(* CODESYS project Traffic_lights.project
   Title: Traffic_lights_ordinary
   Version: 0.0.0.0
   Author: Armin

Project tree, tasks and I/O mapping:
  MyController : TM241CE24T/U, Schneider Electric, order no. TM241CE24T/U, version 4.0.6.18
    application Application
      task MAST (cyclic, interval 20 ms, priority 15, watchdog 100 ms x 1) calls POU, POU_1
      global variables GVL
      Symbols
      program POU [SFC]: Sporedna_active, Sporedna_entry, Glavna_active, Glavna_entry, SveZuto_active, SveZuto_entry, SveZuto_exit, SamoGlavna_entry, SamoGlavna_active, SamoGlavna_exit, SamoSporedna_active, SamoSporedna_entry, SamoSporedna_exit
      program POU_1 [ST]
    DI : Digital Inputs, Schneider Electric, version 4.0.6.18
        input  iwDI_IW0 : WORD  // IW0
        input  ibDI_IB1 : BYTE  // IB1
    DQ : Digital Outputs, Schneider Electric, version 4.0.6.18
        output qwDQ_QW0 : WORD  // QW0
        output qbDQ_QB1 : BYTE  // QB1
    Counters : Counters, Schneider Electric, version 4.0.6.18
    Pulse_Generators : Pulse Generators, Schneider Electric, version 4.0.6.18
    Cartridge_1 : Cartridge, Schneider Electric, version 4.0.6.18
    IO_Bus : IO bus - TM3, Schneider Electric, version 4.0.6.18
    COM_Bus : COM bus, Schneider Electric, version 4.0.6.18
    Ethernet_1 : Ethernet Network, Schneider Electric, version 4.0.6.18
    Serial_Line_1 : Serial line, Schneider Electric, version 4.0.6.18
      SoMachine_Network_Manager : SoMachine-Network Manager, Schneider Electric, version 4.0.0.2
    Serial_Line_2 : Serial line, Schneider Electric, version 4.0.6.18
      Modbus_Manager : Modbus Manager, Schneider Electric, version 4.0.0.2
  XBTGT7340 : XBTGT7340, Schneider Electric, order no. XBTGT7340, version 3.5.3.54
    HMI Application
    COM1
      SoMachine_Network_Manager1 : SoMachine-Network Manager, Schneider Electric, version 4.0.0.2
    COM2
      SoMachine_Network_Manager2 : SoMachine-Network Manager, Schneider Electric, version 4.0.0.2
    Ethernet
      SoMachine_Network_Manager3 : SoMachine-Network Manager, Schneider Electric, version 4.0.0.2
    USB
      SoMachine_Network_Manager4 : SoMachine-Network Manager, Schneider Electric, version 4.0.0.2
  Vijeo Designer Project Container Data
  Vijeo Designer Project Container
*)

// MyController/Application/GVL
VAR_GLOBAL
	sifra: INT;
	stanje: BOOL;
	T1: TP;
	potvrdi: BOOL;
	vratiNaNulu: BOOL;
	
	proba: BOOL;
	noviStart: BOOL;
	noviStop: BOOL;
	
	ispis: INT;
	Glavna_dodatno_vrijeme: INT := 0;
	Sporedna_dodatno_vrijeme: INT := 0;
	
	Vrijeme_glavne_trake: INT := 65;
	Vrijeme_sporedne_trake: INT := 15;
	
	Inicijalno_vrijeme_glavne_trake: INT := 65;
	Inicijalno_vrijeme_sporedne_trake: INT := 15;
	
	Glavna_gornja_granica: INT := 120;
	Glavna_donja_granica: INT := 60;
	
	Sporedna_gornja_granica: INT := 120;
	Sporedna_donja_granica: INT := 12;
	
	Greska_unos_vremena1: BOOL;
	Greska_unos_vremena2: BOOL;
	
	Zuto_FF: RS;
	Zuto_FF_set: BOOL;
	Zuto_FF_reset: BOOL;
	
	save_glavna_vrijeme: INT;
	save_sporedna_vrijeme: INT;
	
	klik_na_glavna_save: BOOL;
	klik_na_sporedna_save: BOOL;
	uso1: BOOL;
	uso2: BOOL;
	proso1: BOOL := 1;
	
	Glavna_FF: RS;
	Glavna_FF_set: BOOL;
	Glavna_FF_reset: BOOL;
	
	Sporedna_FF: RS;
	Sporedna_FF_set: BOOL;
	Sporedna_FF_reset: BOOL;
	
	resetuj: BOOL;
END_VAR

// MyController/Application/POU
PROGRAM POU
VAR
	okidac: BOOL;
	timer: TOF;
	Glavna4_G: BOOL;
	Glavna4_Y: BOOL;
	Glavna4_R: BOOL;
	Glavna4_lijevo_G: BOOL;
	Glavna4_lijevo_Y: BOOL;
	Glavna4_lijevo_R: BOOL;
	Glavna5_G: BOOL;
	Glavna5_Y: BOOL;
	Glavna5_R: BOOL;
	Glavna5_lijevo_G: BOOL;
	Glavna5_lijevo_Y: BOOL;
	Glavna5_lijevo_R: BOOL;
	Sporedna_G: BOOL;
	Sporedna_Y: BOOL;
	Sporedna_R: BOOL;
	Sporedna_blinkanje: BOOL;
	Glavna5_lijevo_blinkanje: BOOL;
	Glavna5_blinkanje: BOOL;
	Glavna4_lijevo_blinkanje: BOOL;
	Glavna4_blinkanje: BOOL;
	Tramvaj: BOOL;
	Glavna5_pjesaci: BOOL;
	Glavna5_pjesaci_preko: BOOL;
	// Trebao bi se ukljuciti odmah po ukljucenju crvenog na tom dijelu, sto nije slucaj u stvarnosti
	Glavna4_pjesaci: BOOL;
	Glavna4_pjesaci_preko: BOOL;
	Sporedna_jug_pjesaci: BOOL;
	// Trebalo bi se odmah ukljuciti cim se ukljuci zeleno na Glavna5, ovako ni pjesaci ni vozaci nisu sigurni ko treba da ide, jer se za zeleno pjesake ceka 4 sekunde od zelenog za vozace
	Sporedna_sjever_pjesaci: BOOL;
	Sve_zuto_blinkanje: BOOL;
END_VAR

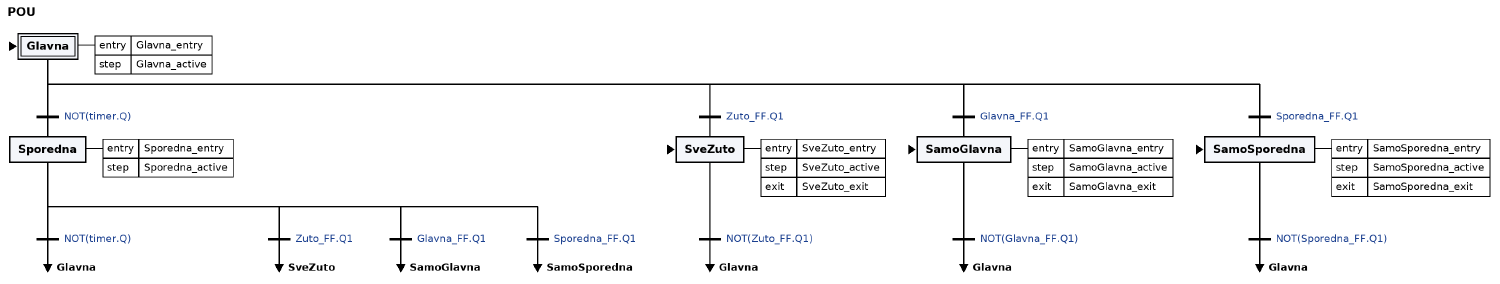
INITIAL_STEP Glavna:
    Glavna_entry(P1);  // entry action
    Glavna_active(N);  // step action
END_STEP
TRANSITION FROM Glavna TO Sporedna
    := NOT(timer.Q);
END_TRANSITION
STEP Sporedna:
    Sporedna_entry(P1);  // entry action
    Sporedna_active(N);  // step action
END_STEP
TRANSITION FROM Sporedna TO Glavna
    := NOT(timer.Q);
END_TRANSITION
TRANSITION FROM Sporedna TO SveZuto
    := Zuto_FF.Q1;
END_TRANSITION
TRANSITION FROM Sporedna TO SamoGlavna
    := Glavna_FF.Q1;
END_TRANSITION
TRANSITION FROM Sporedna TO SamoSporedna
    := Sporedna_FF.Q1;
END_TRANSITION
TRANSITION FROM Glavna TO SveZuto
    := Zuto_FF.Q1;
END_TRANSITION
STEP SveZuto:
    SveZuto_entry(P1);  // entry action
    SveZuto_active(N);  // step action
    SveZuto_exit(P0);  // exit action
END_STEP
TRANSITION FROM SveZuto TO Glavna
    := NOT(Zuto_FF.Q1);
END_TRANSITION
TRANSITION FROM Glavna TO SamoGlavna
    := Glavna_FF.Q1;
END_TRANSITION
STEP SamoGlavna:
    SamoGlavna_entry(P1);  // entry action
    SamoGlavna_active(N);  // step action
    SamoGlavna_exit(P0);  // exit action
END_STEP
TRANSITION FROM SamoGlavna TO Glavna
    := NOT(Glavna_FF.Q1);
END_TRANSITION
TRANSITION FROM Glavna TO SamoSporedna
    := Sporedna_FF.Q1;
END_TRANSITION
STEP SamoSporedna:
    SamoSporedna_entry(P1);  // entry action
    SamoSporedna_active(N);  // step action
    SamoSporedna_exit(P0);  // exit action
END_STEP
TRANSITION FROM SamoSporedna TO Glavna
    := NOT(Sporedna_FF.Q1);
END_TRANSITION

ACTION Sporedna_active:
timer(IN := okidac, PT := LINT_TO_TIME((Vrijeme_sporedne_trake - Inicijalno_vrijeme_sporedne_trake)*1000) + T#15S);
okidac := FALSE;

IF timer.ET > T#2S THEN
	Sporedna_R := 0;
	Sporedna_Y := 0;
	Sporedna_G := 1;
END_IF

IF timer.ET > T#3S THEN
	Glavna5_pjesaci_preko := 1;
	Glavna4_pjesaci_preko := 1;
END_IF

IF timer.ET > LINT_TO_TIME((Vrijeme_sporedne_trake - Inicijalno_vrijeme_sporedne_trake)*1000) + T#4S THEN
	Glavna4_pjesaci := 0;
END_IF

IF timer.ET > LINT_TO_TIME((Vrijeme_sporedne_trake - Inicijalno_vrijeme_sporedne_trake)*1000) + T#8S THEN
	Sporedna_blinkanje := 1;
END_IF

IF timer.ET > LINT_TO_TIME((Vrijeme_sporedne_trake - Inicijalno_vrijeme_sporedne_trake)*1000) + T#12S THEN
	Sporedna_blinkanje := 0;
	Sporedna_G := 0;
	Sporedna_Y := 1;
END_IF

IF timer.ET > LINT_TO_TIME((Vrijeme_sporedne_trake - Inicijalno_vrijeme_sporedne_trake)*1000) + T#13S THEN
	Glavna5_pjesaci_preko := 0;
	Glavna4_pjesaci_preko := 0;
END_IF

IF timer.ET > LINT_TO_TIME((Vrijeme_sporedne_trake - Inicijalno_vrijeme_sporedne_trake)*1000) + T#14S THEN
	Sporedna_Y := 0;
	Sporedna_R := 1;
END_IF
END_ACTION

ACTION Sporedna_entry:
okidac := TRUE;
Sporedna_R := 1;
Sporedna_Y := 1;
END_ACTION

ACTION Glavna_active:
timer(IN := okidac, PT := LINT_TO_TIME((Vrijeme_glavne_trake - Inicijalno_vrijeme_glavne_trake)*1000) + T#65S);
okidac := FALSE;

IF timer.ET > T#2S THEN
	Glavna4_Y := 1;
	Glavna4_lijevo_Y := 1;
END_IF

IF timer.ET > T#4S THEN
	Glavna4_R := 0;
	Glavna4_lijevo_R := 0;
	Glavna4_Y := 0;
	Glavna4_lijevo_Y := 0;
	Glavna4_G := 1;
	Glavna4_lijevo_G := 1;
END_IF

IF timer.ET > T#5S THEN
	Sporedna_jug_pjesaci := 1;
END_IF

IF timer.ET > T#10S THEN
	Glavna5_pjesaci := 0;
END_IF

IF timer.ET > T#13S THEN
	Glavna4_lijevo_blinkanje := 1;
END_IF

IF timer.ET > T#17S THEN
	Glavna4_lijevo_blinkanje := 0;
	Glavna4_lijevo_G := 0;
	Glavna4_lijevo_Y := 1;
END_IF

IF timer.ET > T#20S THEN
	Glavna4_lijevo_Y := 0;
	Glavna4_lijevo_R := 1;
END_IF

IF timer.ET > T#23S THEN
	Glavna5_Y := 1;
END_IF

IF timer.ET > T#25S THEN
	Glavna5_R := 0;
	Glavna5_Y := 0;
	Glavna5_G := 1;
	Tramvaj := 1;
END_IF

IF timer.ET > T#26S THEN
	Sporedna_sjever_pjesaci := 1;
END_IF

IF timer.ET > LINT_TO_TIME((Vrijeme_glavne_trake - Inicijalno_vrijeme_glavne_trake)*1000) + T#33S THEN
	Sporedna_jug_pjesaci := 0;
END_IF

IF timer.ET > LINT_TO_TIME((Vrijeme_glavne_trake - Inicijalno_vrijeme_glavne_trake)*1000) + T#40S THEN
	Glavna4_blinkanje := 1;
	Tramvaj := 0;
	Sporedna_sjever_pjesaci := 0;
END_IF

IF timer.ET > LINT_TO_TIME((Vrijeme_glavne_trake - Inicijalno_vrijeme_glavne_trake)*1000) + T#44S THEN
	Glavna4_blinkanje := 0;
	Glavna4_G := 0;
	Glavna4_Y := 1;
END_IF

IF timer.ET > LINT_TO_TIME((Vrijeme_glavne_trake - Inicijalno_vrijeme_glavne_trake)*1000) + T#47S THEN
	Glavna4_Y := 0;
	Glavna4_R := 1;
END_IF

IF timer.ET > LINT_TO_TIME((Vrijeme_glavne_trake - Inicijalno_vrijeme_glavne_trake)*1000) + T#48S THEN
	Glavna5_lijevo_Y := 1;
	Glavna4_pjesaci := 1;
END_IF

IF timer.ET > LINT_TO_TIME((Vrijeme_glavne_trake - Inicijalno_vrijeme_glavne_trake)*1000) + T#50S THEN
	Glavna5_lijevo_R := 0;
	Glavna5_lijevo_Y := 0;
	Glavna5_lijevo_G := 1;
END_IF

IF timer.ET > LINT_TO_TIME((Vrijeme_glavne_trake - Inicijalno_vrijeme_glavne_trake)*1000) + T#56S THEN
	Glavna5_lijevo_blinkanje := 1;
	Glavna5_blinkanje := 1;
END_IF

IF timer.ET > LINT_TO_TIME((Vrijeme_glavne_trake - Inicijalno_vrijeme_glavne_trake)*1000) + T#60S THEN
	Glavna5_lijevo_blinkanje := 0;
	Glavna5_blinkanje := 0;
	Glavna5_G := 0;
	Glavna5_Y := 1;
	Glavna5_lijevo_G := 0;
	Glavna5_lijevo_Y := 1;
END_IF

IF timer.ET > LINT_TO_TIME((Vrijeme_glavne_trake - Inicijalno_vrijeme_glavne_trake)*1000) + T#63S THEN
	Glavna5_Y := 0;
	Glavna5_R := 1;
	Glavna5_lijevo_Y := 0;
	Glavna5_lijevo_R := 1;
END_IF

IF timer.ET > LINT_TO_TIME((Vrijeme_glavne_trake - Inicijalno_vrijeme_glavne_trake)*1000) + T#64S THEN
	Glavna5_pjesaci := 1;
END_IF
END_ACTION

ACTION Glavna_entry:
okidac := TRUE;
Glavna4_R := 1;
Glavna4_lijevo_R := 1;
Glavna5_R := 1;
Glavna5_lijevo_R := 1;
Sporedna_R := 1;
Glavna5_pjesaci := 1;
END_ACTION

ACTION SveZuto_active:
Glavna4_Y := TRUE;
Glavna4_lijevo_Y := TRUE;
Glavna5_Y := TRUE;
Glavna5_lijevo_Y := TRUE;
Sporedna_Y := TRUE;
Sve_zuto_blinkanje := TRUE;
END_ACTION

ACTION SveZuto_entry:
Glavna4_G := FALSE;
Glavna4_R:= FALSE;
Glavna4_lijevo_G:= FALSE;
Glavna4_lijevo_R:= FALSE;
Glavna5_G:= FALSE;
Glavna5_R:= FALSE;
Glavna5_lijevo_G:= FALSE;
Glavna5_lijevo_R:= FALSE;
Sporedna_G:= FALSE;
Sporedna_R:= FALSE;
Sporedna_blinkanje:= FALSE;
Glavna5_lijevo_blinkanje:= FALSE;
Glavna5_blinkanje:= FALSE;
Glavna4_lijevo_blinkanje:= FALSE;
Glavna4_blinkanje:= FALSE;
Tramvaj:= TRUE;
Glavna5_pjesaci:= FALSE;
Glavna5_pjesaci_preko:= FALSE;
Glavna4_pjesaci:= FALSE;
Glavna4_pjesaci_preko:= FALSE;
Sporedna_jug_pjesaci:= FALSE;
Sporedna_sjever_pjesaci:= FALSE;
END_ACTION

ACTION SveZuto_exit:
Glavna4_Y := FALSE;
Glavna4_lijevo_Y := FALSE;
Glavna5_Y := FALSE;
Glavna5_lijevo_Y := FALSE;
Sporedna_Y := FALSE;
Sve_zuto_blinkanje := FALSE;
Tramvaj := FALSE;
END_ACTION

ACTION SamoGlavna_entry:
Glavna4_Y := FALSE;
Glavna4_R:= FALSE;
Glavna4_lijevo_G:= FALSE;
Glavna4_lijevo_Y:= FALSE;
Glavna5_Y:= FALSE;
Glavna5_R:= FALSE;
Glavna5_lijevo_G:= FALSE;
Glavna5_lijevo_Y:= FALSE;
Sporedna_G:= FALSE;
Sporedna_Y:= FALSE;
Sporedna_blinkanje:= FALSE;
Glavna5_lijevo_blinkanje:= FALSE;
Glavna5_blinkanje:= FALSE;
Glavna4_lijevo_blinkanje:= FALSE;
Glavna4_blinkanje:= FALSE;
Tramvaj:= TRUE;
Glavna5_pjesaci:= FALSE;
Glavna5_pjesaci_preko:= FALSE;
Glavna4_pjesaci:= FALSE;
Glavna4_pjesaci_preko:= FALSE;
Sporedna_jug_pjesaci:= TRUE;
Sporedna_sjever_pjesaci:=TRUE;
END_ACTION

ACTION SamoGlavna_active:
Glavna4_G := TRUE;
Glavna4_lijevo_R := TRUE;
Glavna5_G := TRUE;
Glavna5_lijevo_R := TRUE;
Sporedna_R := TRUE;
END_ACTION

ACTION SamoGlavna_exit:
Glavna4_G := FALSE;
Glavna4_lijevo_R := FALSE;
Glavna5_G := FALSE;
Glavna5_lijevo_R := FALSE;
Sporedna_R := FALSE;
Sporedna_jug_pjesaci:= FALSE;
Sporedna_sjever_pjesaci:= FALSE;
Tramvaj:= FALSE;
END_ACTION

ACTION SamoSporedna_active:
Glavna4_R := TRUE;
Glavna4_lijevo_R := TRUE;
Glavna5_R := TRUE;
Glavna5_lijevo_R := TRUE;
Sporedna_G := TRUE;
END_ACTION

ACTION SamoSporedna_entry:
Glavna4_G := FALSE;
Glavna4_Y:= FALSE;
Glavna4_lijevo_G:= FALSE;
Glavna4_lijevo_Y:= FALSE;
Glavna5_G:= FALSE;
Glavna5_Y:= FALSE;
Glavna5_lijevo_G:= FALSE;
Glavna5_lijevo_Y:= FALSE;
Sporedna_Y:= FALSE;
Sporedna_R:= FALSE;
Sporedna_blinkanje:= FALSE;
Glavna5_lijevo_blinkanje:= FALSE;
Glavna5_blinkanje:= FALSE;
Glavna4_lijevo_blinkanje:= FALSE;
Glavna4_blinkanje:= FALSE;
Tramvaj:= FALSE;
Glavna5_pjesaci:= TRUE;
Glavna5_pjesaci_preko:= TRUE;
Glavna4_pjesaci:= TRUE;
Glavna4_pjesaci_preko:= TRUE;
Sporedna_jug_pjesaci:= FALSE;
Sporedna_sjever_pjesaci:= FALSE;
END_ACTION

ACTION SamoSporedna_exit:
Glavna4_R := FALSE;
Glavna4_lijevo_R := FALSE;
Glavna5_R := FALSE;
Glavna5_lijevo_R := FALSE;
Sporedna_G := FALSE;
Glavna5_pjesaci:= FALSE;
Glavna5_pjesaci_preko:= FALSE;
Glavna4_pjesaci:= FALSE;
Glavna4_pjesaci_preko:= FALSE;
END_ACTION

END_PROGRAM

// MyController/Application/POU_1
PROGRAM POU_1
VAR
	akta: BOOL;
	nePotvrdi: INT;
	start: BOOL;
	IN: BOOL;
	noviStop: BOOL;
	TpumpaOn1: INT;
	TpumpaOn2: INT;
END_VAR

VAR_INPUT
	PT: TIME;
	noviStartOR: BOOL;
END_VAR

IF (sifra = 1234) THEN
	stanje := TRUE;
END_IF
IF (sifra <> 1234) THEN
	stanje := FALSE;
END_IF

IF(vratiNaNulu) THEN
	sifra := 0;
END_IF

T1(IN := (potvrdi AND (NOT stanje)), PT := T#11S);
IF (T1.ET > T#10S) THEN
	sifra := 1234;
END_IF

ispis := 10 - TIME_TO_INT(T1.ET)/1000;

IF (Vrijeme_glavne_trake < Glavna_donja_granica) OR (Vrijeme_glavne_trake > Glavna_gornja_granica) THEN
	Greska_unos_vremena1 := TRUE;
ELSE
	Greska_unos_vremena1 := FALSE;
END_IF

IF (Vrijeme_sporedne_trake < Sporedna_donja_granica) OR (Vrijeme_sporedne_trake > Sporedna_gornja_granica) THEN
	Greska_unos_vremena2 := TRUE;
ELSE
	Greska_unos_vremena2 := FALSE;
END_IF

IF resetuj THEN
	Vrijeme_glavne_trake := Inicijalno_vrijeme_glavne_trake;
	Vrijeme_sporedne_trake := Inicijalno_vrijeme_sporedne_trake;
END_IF

Zuto_FF(SET := Zuto_FF_set, RESET1 := Zuto_FF_reset);
Glavna_FF(SET := Glavna_FF_set, RESET1 := Glavna_FF_reset);
Sporedna_FF(SET := Sporedna_FF_set, RESET1 := Sporedna_FF_reset);

END_PROGRAM
